Fanuc KAREL source: kb00142.KL

-- PROVISIONAL review KL for V1013-1; original PC SHA256 993c78db8878de6424960f594e0c8c03fe6ce261e033f63cbdec13f419e78187
-- Incomplete behavior may be omitted. Consult companion uncertainty JSON. Do not deploy.
PROGRAM KB00142
%NOLOCKGROUP
BEGIN
  -- UNRESOLVED_PC offsets 5-14; opcodes 3F,75
  -- UNRESOLVED_PC offsets 19-26; opcodes 9D,23
  -- UNRESOLVED_PC offsets 31-38; opcodes 9D,23
  -- UNRESOLVED_PC offsets 43-50; opcodes 9D,23
  -- UNRESOLVED_PC offsets 55-85; opcodes 27,22,2A,22,22,22,31
  -- UNRESOLVED_PC offsets 90-94; opcodes 7F
END KB00142
